FUNCTION_BLOCK FB_2_ROB_MANIP EXTENDS FB_1_ROB IMPLEMENTS ITF_2_Manip

VAR_INPUT
	Tool: FB_1_Tool;
	bEnableCommunication : BOOL := TRUE;
END_VAR

VAR_OUTPUT
	visStatus: stVisStatusManip;
END_VAR
VAR


	
	//TODO What is this for?
	_command : ST_RobotCommand;
	_commandState : E_RobotCommandState := E_RobotCommandState.Idle;
	_commandErrorId : UDINT;
	_nextExecuteId : UDINT := 1;		
END_VAR

ACTION CYCLIC_MANIP:
CYCLIC_ROB();

visStatus.State:=eStatus;
visStatus.Mode:=eModus;
visStatus.isMoving:=RobotMoving;
visStatus.isReady:=RobotReady;
visStatus.isConnected:=CommunicationReady;
// 	isLocked: BOOL;
// visStatus.isBusy:=;
visStatus.isInCollision:=InCollision;
visStatus.hasError:=Messenger.HasActivError;
visStatus.TCPPosition:=ActualTcpPose;
END_ACTION

{warning 'Add method implementation '}
METHOD Home : UINT


VAR
	Config: stBA_Settings;
END_VAR


Home:= BA_Handler(Cmd:=eBA.Home,Settings:=Config);
END_METHOD

{warning 'Override with your own Method in final FB'}
  PROPERTY IsHomePosition : BOOL
GET
END_GET
END_PROPERTY

METHOD MoveJoint : UINT
VAR_INPUT
    Target : stTarget;
	Velocity: REAL;
END_VAR

VAR
	Config: stBA_Settings;
END_VAR
Config.Velocity:=Velocity;
Config.Target:=Target;


MoveJoint := BA_Handler(Cmd:=eBA.MoveJ,Settings:=Config); //HAndler returns a UINT ID of the BA
END_METHOD


METHOD MoveJointRelative : UINT
VAR_INPUT
    Target : stTarget;
	Velocity: REAL;
END_VAR

VAR
	Config: stBA_Settings;
END_VAR
Config.Velocity:=Velocity;
Config.Target:=Target;


MoveJointRelative:= BA_Handler(Cmd:=eBA.MoveJRelativ,Settings:=Config);
END_METHOD

METHOD MoveLinear : UINT
VAR_INPUT
	Target	: stTarget;
	Velocity: REAL;
END_VAR

VAR
	Config: stBA_Settings;
END_VAR
Config.Velocity:=Velocity;
Config.Target:=Target;


MoveLinear:= BA_Handler(Cmd:=eBA.MoveL,Settings:=Config);
END_METHOD

METHOD MoveLinearRelative : UINT
VAR_INPUT
    Offset : stPoseGeneral;
	Velocity: REAL;
END_VAR

VAR
	Config: stBA_Settings;
END_VAR
Config.Velocity:=Velocity;
Config.Pose:=Offset;


MoveLinearRelative:= BA_Handler(Cmd:=eBA.MoveL,Settings:=Config);
END_METHOD

METHOD SetDO : UINT
VAR_INPUT
    nOutput : UINT;
    bValue : BOOL;
END_VAR

VAR
	Config: stBA_Settings;
END_VAR
Config.Pin:=nOutput;
Config.bValue:=bValue;


SetDO:= BA_Handler(Cmd:=eBA.SetDO,Settings:=Config);
END_METHOD

{warning 'Override with your own Method in final FB'}
PROPERTY TargetReached : BOOL
GET
TargetReached := _commandState = E_RobotCommandState.Done;
END_GET
END_PROPERTY

END_FUNCTION_BLOCK

(* stored: Version 1.1.0.1, ProductVersion 3.1.4026.18
   POU FB_2_ROB_MANIP: Id {21b924b4-0fb6-46ff-9fb7-f679235d19bb}, SpecialFunc None
   Folder MotionControl: Id {fc8c0aca-629b-4848-a20d-78e9ce6e9fda}
   Action CYCLIC_MANIP: Id {c5ea77dd-14da-4015-9108-0744e50afbab}
   Method Home: Id {332921a2-9f70-499b-943d-00519405a468}
   Property IsHomePosition: Id {0f2fd807-aeed-459c-9c2b-f2325fe045e7}
   Get Get: Id {cc381350-4b9b-4a45-a9c1-b7537b47d8d7}
   Method MoveJoint: Id {9e0f1a2b-3c4d-4e5f-8a6b-7c8d9e0f1a2b}
   Method MoveJointRelative: Id {d4d7d377-1aa7-4fc3-9e59-f55d00fe8d35}
   Method MoveLinear: Id {af96fe73-c0fb-4331-8a41-58ccd3cdc293}
   Method MoveLinearRelative: Id {bc2132e6-39c8-42b1-8dcb-1b232e67fc7a}
   Method SetDO: Id {1b1484e8-2eba-4b5a-9bc9-3e9f0cf73af2}
   Property TargetReached: Id {2237dc56-6e31-4e2f-87fb-158a23ca2344}
   Get Get: Id {fa9b9558-e97e-4d6d-afa4-8757f8a89ab1} *)
